// TIA Portal V18 export
FUNCTION "ST10_ChangeOver" : Void   // FC1008, LAD
{ S7_Optimized_Access := 'FALSE' }
// stored: AutoNumber false, SetENOAutomatically false
   VAR_TEMP
      sString : String[50];
      FixtureNumber : Int;
      FixtureIndex : Int;
      tRET_VAL : Int;
   END_VAR
BEGIN

REGION Network 1: Recipe Active
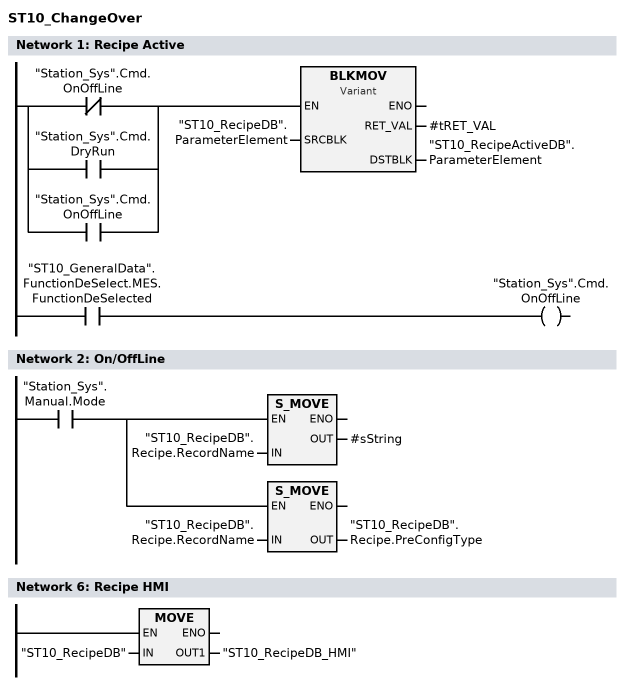
   RUNG wire#powerrail
      I_Contact( "Station_Sys".Cmd.OnOffLine )
      wire#w1
      { S7_Templates := "blk_type := Variant" } BLKMOV(SRCBLK := "ST10_RecipeDB".ParameterElement, RET_VAL => #tRET_VAL, DSTBLK => "ST10_RecipeActiveDB".ParameterElement)
   END_RUNG
   RUNG wire#powerrail
      Contact( "Station_Sys".Cmd.DryRun )
   END_RUNG wire#w1
   RUNG wire#powerrail
      Contact( "Station_Sys".Cmd.OnOffLine )
   END_RUNG wire#w1
   RUNG wire#powerrail
      Contact( "ST10_GeneralData".FunctionDeSelect.MES.FunctionDeSelected )
      Coil( "Station_Sys".Cmd.OnOffLine )
   END_RUNG
   // the same network as SCL:
   IF NOT "Station_Sys".Cmd.OnOffLine OR "Station_Sys".Cmd.DryRun OR "Station_Sys".Cmd.OnOffLine THEN
       #tRET_VAL := BLKMOV(SRCBLK := "ST10_RecipeDB".ParameterElement,
                           DSTBLK => "ST10_RecipeActiveDB".ParameterElement);
   END_IF;
   "Station_Sys".Cmd.OnOffLine := "ST10_GeneralData".FunctionDeSelect.MES.FunctionDeSelected;
END_REGION

REGION Network 2: On/OffLine
   RUNG wire#powerrail
      Contact( "Station_Sys".Manual.Mode )
      wire#w1
      S_Move(in := "ST10_RecipeDB".Recipe.RecordName, out => #sString)
   END_RUNG
   RUNG wire#w1
      S_Move(in := "ST10_RecipeDB".Recipe.RecordName, out => "ST10_RecipeDB".Recipe.PreConfigType)
   END_RUNG
   // the same network as SCL:
   IF "Station_Sys".Manual.Mode THEN
       #sString := "ST10_RecipeDB".Recipe.RecordName;
       "ST10_RecipeDB".Recipe.PreConfigType := "ST10_RecipeDB".Recipe.RecordName;
   END_IF;
END_REGION

NETWORK
TITLE = 换型功能块调用 / Transposition function block call
//"ST10_RecipeDB".Recipe.PreConfigType    AUTO CONFIG, When PLC activate change over, Set Recipe data record Tags
//"ST10_RecipeDB".ParameterElement.TypeName    HMI MANUAL CONFIG, HMI Recipe data record element:Product_type
//HMI Recipe data record element Product_type set value must be same with HMI Recipe data record Name

      A     "ChangeOver_DB".Global.ChangeOverActive;
      A     "Station_Sys".Auto.Mode;
      =     "ST10_RecipeDB".Recipe.Trigger;

      CALL  "ChangeOver"
      ( iCheckType      := "ST10_RecipeDB".ParameterElement.TypeName,
        "iPulse*500ms"  := "Sys".COM.FlashTime500mS,
        iReset          := "Station_Sys".Cmd.Reset,
        Ret_Val         := "ST10_RecipeDB".Recipe.Ret,
        oPulse          := "ST10_RecipeDB".Recipe.Pulse,
        oEqual          := "ST10_RecipeDB".Recipe.Equal,  // CheckType=PreConfigType, indicate ChangerOver successfully
        ioPreConfigType := "ST10_RecipeDB".Recipe.PreConfigType,
        ioCurrentName   := "ST10_RecipeDB".Recipe.RecordName,
        iotime          := "ST10_RecipeDB".Recipe."time",
        ioTrigger       := "ST10_RecipeDB".Recipe.Trigger,
        ioPosEdg        := "ST10_RecipeDB".Recipe.PosEdg,
        ioAlarm         := "ST10_RecipeDB".Recipe.Alarm,
        ioPls           := "ST10_RecipeDB".Recipe.Pls
      );




REGION Network 4 (SCL): Fixture换型工装 / Fixture Changing fixture
   //Fixture 1 输入轴换型X轴工装
   //工装检测屏蔽条件
   "ST10_GeneralData".FixtureIDCheck[1].FixtureCheckUnEnable := 0;

   //工装检测传感器赋值

   "ST10_GeneralData".FixtureIDCheck[1].FixtureIDCheckValue.%X0 := 0;
   "ST10_GeneralData".FixtureIDCheck[1].FixtureIDCheckValue.%X1 := 0;
   "ST10_GeneralData".FixtureIDCheck[1].FixtureIDCheckValue.%X2 := 0;
   "ST10_GeneralData".FixtureIDCheck[1].FixtureIDCheckValue.%X3 := 0;
   "ST10_GeneralData".FixtureIDCheck[1].FixtureIDCheckValue.%X4 := 0;
   "ST10_GeneralData".FixtureIDCheck[1].FixtureIDCheckValue.%X5 := 0;
   "ST10_GeneralData".FixtureIDCheck[1].FixtureIDCheckValue.%X6 := 0;
   "ST10_GeneralData".FixtureIDCheck[1].FixtureIDCheckValue.%X7 := 0;
END_REGION

REGION Network 5 (SCL): FixtureID Check Call
   //循环数量为工装检测的数量

   #FixtureNumber := 1;

   //工装检测功能块调用

   #FixtureIndex := 1;

   FOR #FixtureIndex := 1 TO #FixtureNumber DO

       "fcFixtureCheck"(iRecipeSetValue := "ST10_RecipeDB".ParameterElement.FixtureID[#FixtureIndex],
                        FixtureIDCheck := "ST10_GeneralData".FixtureIDCheck[#FixtureIndex]);

   END_FOR;
END_REGION

REGION Network 6: Recipe HMI
   RUNG wire#powerrail
      Move(in := "ST10_RecipeDB", out1 => "ST10_RecipeDB_HMI")
   END_RUNG
   // the same network as SCL:
   "ST10_RecipeDB_HMI" := "ST10_RecipeDB";
END_REGION
END_FUNCTION
